// Jidien Kachu Edited in 2025/09/25
FUNCTION_BLOCK FB_WareHouseWithRobotMove_V2 EXTENDS FB_ObjectBase_V2 IMPLEMENTS IBasicElement
VAR_INPUT
    Robot     : REFERENCE TO FB_FanucRobot_Basic;
    WareHouse : REFERENCE TO FB_WareHouse;
   // Command   : ST_WareHouseWithRobotMove_Command;
    Info	  : st_AutoSixAxisWarehouseParameter;
	Stop	  : BOOL;
	//Edited by Jidien Kachu in 2025/09/25
	iSetRetryCnt	: UINT := 10;
END_VAR
VAR_OUTPUT
  // Status : ST_WareHouseWithRobotMove_Status;
END_VAR
VAR
	_Abort		: BOOL;
	strStatus	: STRING;
	uiResumeStep : UINT;
	ClampA_WareHouseCoordinates : ST_WareHouseCoordinates;
    ClampB_WareHouseCoordinates : ST_WareHouseCoordinates;
	UseA 	: BOOL;
	UseB	: BOOL;
	TargetWarehouse : E_WareHouse;
	Get 	:BOOL;
	tonTimeout		:TON;
	bTimeOutIN			   : BOOL;
	tonRobotTimeout		:TON;
	bRobotTimeoutIN			   : BOOL;
	_UniqueErrorCode :STRING;
	PreviousStrStatus : STRING;
	PreviousErrorCode : STRING;
	//Edited by Jidien Kachu in 2025/09/25
	iActRetryCnt	: UINT;
	uiBothStep : UINT;
	uiLastBothStep : UINT;
END_VAR

SUPER^.A10_StateControl();
A00_BasicUnits();

ACTION A00_BasicUnits:
tonTimeOut(IN:= bTimeOutIN AND NOT THIS^.Stop, PT:=T#30S);
tonRobotTimeout(IN:= bRobotTimeoutIN AND NOT THIS^.Stop,PT:=T#60S);
ErrorID :=2400;
END_ACTION

METHOD M_CheckCommand : BOOL // True : Command is useful
VAR_INPUT
END_VAR
VAR
	
END_VAR
// Check command paremeter is correct

IF NOT Info.Warehouse_A AND NOT Info.Warehouse_B THEN
	strStatus:='Wrong command , No warehouse selected';
	M_CheckCommand:=FALSE;
	RETURN;
ELSIF  Info.Warehouse_A AND  Info.Warehouse_B THEN
	strStatus:='Wrong command , Both warehouses selected';
	M_CheckCommand:=FALSE;
	RETURN;
ELSIF	Info.Warehouse_A THEN
	TargetWarehouse:=E_WareHouse.WareHouseA;
ELSIF	Info.Warehouse_B THEN
	TargetWarehouse:=E_WareHouse.WareHouseB;
END_IF

IF Info.Get_A <> Info.Get_B THEN
	strStatus:='Wrong command ,GetA not match to GetB';
	M_CheckCommand:=FALSE;
	RETURN;
	ELSE
		
	Get :=Info.Get_A;
END_IF


CASE LREAL_TO_INT(Info.Layer_A) OF

1,2,3,4,5,6,7,8,9,10:
	//Normal
	// Layer A in correct range
	IF ((Info.Slide_A < 1) OR (Info.Slide_A > 20)) THEN
		strStatus := 'Command error : Clamp A target slide out of range';
		M_CheckCommand:=FALSE;
		RETURN;
	ELSE
		ClampA_WareHouseCoordinates.Layer:=LREAL_TO_INT(Info.Layer_A);
		ClampA_WareHouseCoordinates.Slide:=LREAL_TO_INT(Info.Slide_A);
   
		UseA:=TRUE;	
	END_IF
	
99:
	UseA:=FALSE;
ELSE
	 strStatus := 'Command error : Clamp A target layer out of range.';
	 M_CheckCommand:=FALSE;
	 RETURN;
END_CASE


CASE LREAL_TO_INT(Info.Layer_B) OF

1,2,3,4,5,6,7,8,9,10:
//Normal
	// Layer A in correct range
	IF ((Info.Slide_B < 1) OR (Info.Slide_B > 20)) THEN
		strStatus := 'Command error : Clamp B target slide out of range';
		M_CheckCommand:=FALSE;
		RETURN;
	ELSE
		ClampB_WareHouseCoordinates.Layer:=LREAL_TO_INT(Info.Layer_B);
		ClampB_WareHouseCoordinates.Slide:=LREAL_TO_INT(Info.Slide_B);
		UseB:=TRUE;	
	END_IF
	
99:
		UseB:=FALSE;
ELSE
	 strStatus := 'Command error : Clamp B target layer out of range.';
	 M_CheckCommand:=FALSE;
	 RETURN;
END_CASE


M_CheckCommand:=TRUE;
END_METHOD

METHOD M_CheckUnitsNotBusy : BOOL
VAR_INPUT
END_VAR
M_CheckUnitsNotBusy := true;
END_METHOD

METHOD M_CheckUnitsReady : BOOL
VAR_INPUT
END_VAR
M_CheckUnitsReady := true;
END_METHOD

METHOD  M_STATE_ABORTED
VAR_INPUT
END_VAR
ERROR :=TRUE;
Busy    := FALSE;
Aborted := TRUE;
Status := strStatus;
UniqueErrorCode:=_UniqueErrorCode;
IF NOT Execute THEN
	eSTATE:=STATE_RESETTING;
END_IF

IF Execute AND Reset THEN 
	PreviousStrStatus := strStatus;
	PreviousErrorCode := _UniqueErrorCode;
	uiExecutingStep :=uiResumeStep;
	eSTATE:=STATE_EXECUTING;
	
	iActRetryCnt := iActRetryCnt + 1; //Edited by Jidien Kachu in 2025/09/25
	ERROR :=FALSE;
	Aborted := FALSE;
	uiBothStep := uiLastBothStep;
END_IF
END_METHOD

METHOD  M_STATE_ABORTING
VAR_INPUT
END_VAR
CASE uiAbortingStep OF
	0 :
		uiAbortingStep:=9999;
		bTimeOutIN:=FALSE;
		bRobotTimeoutIN :=FALSE;
		IF strStatus = PreviousStrStatus THEN
			_UniqueErrorCode :=PreviousErrorCode;
		END_IF
		_Abort :=FALSE;
		(*=====Edited by Jidien Kachu in 2025/09/25=====*)
		Robot.M_ResetAllCommand();
		WareHouse.M_ResetReloadBox();
		WareHouse.M_ResetFeedInBox();
		(*==============================================*)
	9999:	_AbortCompleted:=TRUE;
END_CASE

IF _AbortCompleted THEN	
	eSTATE :=STATE_ABORTED;
END_IF
END_METHOD

METHOD  M_STATE_DONE
VAR_INPUT
END_VAR
Busy := FALSE;
Done := TRUE;
IF NOT Execute THEN
    eState := STATE_RESETTING;
END_IF
END_METHOD

METHOD  M_STATE_DORMANT
VAR_INPUT
END_VAR
// Clear FB output
Busy            := FALSE;
Done            := FALSE;
Aborted         := FALSE;
Error           := FALSE;
ErrorID         := 0;
Status          := '';
_ResetCompleted := FALSE;
_Error          := FALSE;
_Executed       := FALSE;
strStatus :='No Error';
bTimeOutIN :=FALSE;
bRobotTimeoutIN :=FALSE;
uiExecutingStep :=uiResettingStep :=uiResumeStep :=0;
PreviousStrStatus			 :='';
PreviousErrorCode			 :='';

// Wait Execute command
IF Execute THEN
    eState := STATE_EXECUTING;
END_IF
END_METHOD

METHOD  M_STATE_ERROR
VAR_INPUT
END_VAR
ERROR   :=TRUE;
Busy	:=FALSE;
Status := strStatus;
UniqueErrorCode:=_UniqueErrorCode;
IF NOT Execute THEN	
eSTATE:=STATE_RESETTING;
END_IF
END_METHOD

METHOD  M_STATE_EXECUTING
VAR_INPUT
END_VAR
VAR_INST
	BoxReady_1st : BOOL;
	BoxReady_2nd : BOOL;  
    
    ClampA_WareHouseCoordinates : ST_WareHouseCoordinates;
    ClampB_WareHouseCoordinates : ST_WareHouseCoordinates;
	

	
END_VAR
VAR
	
END_VAR
// Set Busy active edit by johnson
Busy := TRUE;
(*IF THIS^.Stop THEN // Pending the timeout when Stop signal occur
	bTimeOutIN :=FALSE;
	bRobotTimeoutIN :=FALSE;
END_IF*)
// Service Process
CASE uiExecutingStep OF
	0:
        // Clear variable
       
        bTimeOutIN :=FALSE;
//        uiBothStep := 0;
		uiLastBothStep := 0; //Edited by Jidien Kachu in 2025/10/09
		BoxReady_1st := 0;
		BoxReady_2nd := 0;
        // Check command
        IF M_CheckCommand() THEN
            uiExecutingStep := 10;
		ELSE
			_Error:=TRUE;
        END_IF
		iActRetryCnt := 0; //Edited by Jidien Kachu in 2025/09/25
    10:
        // Start process, check units first
        IF M_CheckUnitsReady() THEN
            uiExecutingStep := 20;
        END_IF
    20:
        // CHeck units not busy state
        IF M_CheckUnitsNotBusy() THEN
            uiExecutingStep := 1000;
        END_IF
   
	1000:   
			// Read  Warehouse coordinate
			ClampA_WareHouseCoordinates := THIS^.ClampA_WareHouseCoordinates;
            ClampB_WareHouseCoordinates := THIS^.ClampB_WareHouseCoordinates;     
			IF UseA AND NOT UseB THEN
				//Only clampA
				uiExecutingStep := 10000;
			ELSIF NOT UseA AND UseB THEN
				//Only ClampB 
				uiExecutingStep := 20000;
			ELSIF UseA AND UseB THEN
				//Both Clamps
				uiExecutingStep := 30000;		
			END_IF
       
    10000: // Only ClampA 
        IF NOT Robot._DI1.Done THEN
            // Read ClampA Warehouse coordinate
            ClampA_WareHouseCoordinates := THIS^.ClampA_WareHouseCoordinates;
			
			IF Get THEN// Prepare Box
				//Pick Box
				 WareHouse.M_StartReloadBox(WareHouseSelect := TargetWarehouse, WarehouseCoordinates := ClampA_WareHouseCoordinates);

           		 // Check Box reload completed
           		 IF WareHouse.bReloadBox_Completed THEN
           	     BoxReady_1st := TRUE;
          		  END_IF
				  // Robot Warehouse move
           		 Robot.M_StartWareHousePickUpBox_ClampA(WareHouseSelect := TargetWarehouse,
                                                   Info            := ClampA_WareHouseCoordinates,
                                                   BoxReady_1st    := BoxReady_1st);
//				bTimeOutIN:=TRUE;
				IF tonTimeout.Q THEN
					_Error:=TRUE;
					strStatus:='Clamp A reolad box timeout';
				END_IF
				  
			ELSE
					//Place Box
					WareHouse.M_StartFeedInBox(WareHouseSelect := TargetWarehouse, WarehouseCoordinates := ClampA_WareHouseCoordinates);

           			 // Check Box reload completed
           			 IF WareHouse.bFeedInBox_Completed THEN
               			 BoxReady_1st := TRUE;
          		 	 END_IF				
					           
			 	Robot.M_StartWareHousePlaceBox_ClampA(WareHouseSelect := TargetWarehouse,
                                                   Info            := ClampA_WareHouseCoordinates,
                                                   BoxReady_1st    := BoxReady_1st);
            	
//				bTimeOutIN:=TRUE;
				IF tonTimeout.Q THEN
					_Error:=TRUE;
					strStatus:='Clamp A Feedin box timeout';
				END_IF
           END_IF
        ELSE
            uiExecutingStep := 10080;
        END_IF
		
		bRobotTimeoutIN :=TRUE;
		IF tonRobotTimeout.Q THEN
			(*=====Edited by Jidien Kachu in 2025/09/25=====*)
			IF iActRetryCnt = iSetRetryCnt THEN
				_Error:=TRUE;
			ELSE
				_Abort := TRUE;
				uiAbortingStep := 0;
			END_IF
			
			(*==============================================*)
			strStatus:='Clamp A  robot timeout';
		END_IF
		
    10080:
        Robot.M_ResetAllCommand(); // Clear command and go to place box
		bTimeOutIN :=FALSE;
		bRobotTimeoutIN :=FALSE;
        IF NOT Robot._DI1.Done THEN
            uiExecutingStep := 99000; 
        END_IF
    
    
   20000: // Only ClampB
        IF NOT Robot._DI1.Done THEN
            			
			IF Get THEN// Prepare Box
				//Pick Box
				 WareHouse.M_StartReloadBox(WareHouseSelect := TargetWarehouse, WarehouseCoordinates := ClampB_WareHouseCoordinates);

           		 // Check Box reload completed
           		 IF WareHouse.bReloadBox_Completed THEN
           	     BoxReady_2nd := TRUE;
          		  END_IF
				  // Robot Warehouse move
           		 Robot.M_StartWareHousePickUpBox_ClampB(WareHouseSelect := TargetWarehouse,
                                                   Info            := ClampB_WareHouseCoordinates,
                                                   BoxReady_2nd    := BoxReady_2nd);

//				bTimeOutIN:=TRUE;
				IF tonTimeout.Q THEN
					_Error:=TRUE;
					strStatus:='Clamp B Reload box timeout';
				END_IF
			ELSE
					//Place Box
					WareHouse.M_StartFeedInBox(WareHouseSelect := TargetWarehouse, WarehouseCoordinates := ClampB_WareHouseCoordinates);

           			 // Check Box reload completed
           			 IF WareHouse.bFeedInBox_Completed THEN
               			 BoxReady_2nd := TRUE;
          		 	 END_IF				
					           
			 	Robot.M_StartWareHousePlaceBox_ClampB (WareHouseSelect := TargetWarehouse,
                                                   Info            := ClampB_WareHouseCoordinates,
                                                   BoxReady_2nd    := BoxReady_2nd);
//            	bTimeOutIN:=TRUE;
				IF tonTimeout.Q THEN
					_Error:=TRUE;
					strStatus:='Clamp B Feedin box timeout';
				END_IF
           END_IF
        ELSE
            uiExecutingStep := 20080;
        END_IF
		
		bRobotTimeoutIN :=TRUE;
		IF tonRobotTimeout.Q THEN
			(*=====Edited by Jidien Kachu in 2025/09/25=====*)
			IF iActRetryCnt = iSetRetryCnt THEN
				_Error:=TRUE;
			ELSE
				_Abort := TRUE;
				uiAbortingStep := 0;
			END_IF
			(*==============================================*)
			strStatus:='Clamp B Robot timeout';
		END_IF
		
    20080:
        Robot.M_ResetAllCommand(); // Clear command and go to place box
		bTimeOutIN :=FALSE;
		bRobotTimeoutIN :=FALSE;

        IF NOT Robot._DI1.Done THEN
            uiExecutingStep := 99000; 
        END_IF
		
    30000: // Both Clamps
        		
		IF Get THEN //BOth clamps pick
        CASE uiBothStep OF
            0: // ClampA target slide move the box to front side
                WareHouse.M_StartReloadBox(WareHouseSelect      := TargetWarehouse,
                                           WarehouseCoordinates := ClampA_WareHouseCoordinates);
				
				bTimeOutIN :=TRUE;
				IF tonTimeout.Q THEN
					(*=====Edited by Jidien Kachu in 2025/09/25=====*)
					IF iActRetryCnt = iSetRetryCnt THEN
						_Error:=TRUE;
					ELSE
						_Abort := TRUE;
						uiAbortingStep := 0;
					END_IF
					(*==============================================*)
					strStatus:='Clamp A reload timeout';
				END_IF
               
                IF WareHouse.bReloadBox_Completed THEN
					bTimeOutIN :=FALSE;
                    BoxReady_1st     := TRUE;
                    uiBothStep := 10;
                END_IF

            10: // wait Robot Allow continue
			 		WareHouse.M_ResetReloadBox();
                IF Robot._DI1.Notification // AND
//                    NOT
//                    WareHouse._stWarehouseList.ASide_Layers[ClampA_WareHouseCoordinates.Layer].stStatus.bSlides[ClampA_WareHouseCoordinates.Slide]
                    THEN
                   
					
                    IF NOT WareHouse.bReloadBox_Completed THEN					
               
                        uiBothStep := 15;
                    END_IF

                END_IF
			15:	IF NOT WareHouse._stWarehouseList.ASide_Layers[ClampA_WareHouseCoordinates.Layer].stStatus.bSlides[ClampA_WareHouseCoordinates.Slide] THEN
					 uiBothStep := 20;	
				 END_IF
				 
            20: // ClampB target slide move the box to front slide
                WareHouse.M_StartReloadBox(WareHouseSelect := TargetWarehouse, WarehouseCoordinates := ClampB_WareHouseCoordinates);
				bTimeOutIN :=TRUE;
                IF WareHouse.bReloadBox_Completed THEN
					bTimeOutIN :=FALSE;
                    BoxReady_2nd     := TRUE;
                    uiBothStep := 99;
                END_IF
				IF tonTimeout.Q THEN
					(*=====Edited by Jidien Kachu in 2025/09/25=====*)
					IF iActRetryCnt = iSetRetryCnt THEN
						_Error:=TRUE;
					ELSE
						_Abort := TRUE;
						uiAbortingStep := 0;
						uiLastBothStep := 20;
					END_IF
					(*==============================================*)
					strStatus:='Clamp B reload timeout';
				END_IF
				
				
            99:
				WareHouse.M_ResetReloadBox();
        // wait reset
        END_CASE

        Robot.M_StartWareHousePickUpBox_ClampBoth(WareHouseSelect := TargetWarehouse,
                                                  ClampA_Info     := ClampA_WareHouseCoordinates,
                                                  ClampB_Info     := ClampB_WareHouseCoordinates,
                                                  BoxReady_1st    := BoxReady_1st,
                                                  BoxReady_2nd    := BoxReady_2nd);
												  
		bRobotTimeoutIN :=TRUE;
		IF tonRobotTimeout.Q THEN
			(*=====Edited by Jidien Kachu in 2025/09/25=====*)
			IF iActRetryCnt = iSetRetryCnt THEN
				_Error:=TRUE;
			ELSE
				_Abort := TRUE;
				uiAbortingStep := 0;
			END_IF
			(*==============================================*)
			strStatus:='Robot timeout';
		END_IF
		ELSE
		  CASE uiBothStep OF
			  
			   0: // ClampA target slide move the box to front side
                WareHouse.M_StartFeedInBox(WareHouseSelect      := TargetWarehouse,
                                           WarehouseCoordinates := ClampA_WareHouseCoordinates);

               bTimeOutIN :=TRUE;
                IF WareHouse.bFeedInBox_Completed THEN
					bTimeOutIN :=FALSE;
                    BoxReady_1st     := TRUE;
                    uiBothStep := 10;
                END_IF
				IF tonTimeout.Q THEN
					(*=====Edited by Jidien Kachu in 2025/09/25=====*)
					IF iActRetryCnt = iSetRetryCnt THEN
						_Error:=TRUE;
					ELSE
						_Abort := TRUE;
						uiAbortingStep := 0;
					END_IF
					(*==============================================*)
					strStatus:='Clamp A Feedin timeout';
				END_IF

            10: // wait Robot Allow continue
					WareHouse.M_ResetFeedInBox();
                 IF Robot._DI1.Notification //AND
                     
//                    WareHouse._stWarehouseList.ASide_Layers[ClampA_WareHouseCoordinates.Layer].stStatus.bSlides[ClampA_WareHouseCoordinates.Slide]
                    THEN
                    

                    IF NOT WareHouse.bFeedInBox_Completed THEN
                        uiBothStep := 15;
                    END_IF

                END_IF
			15:  
				uiBothStep := 20;
			
            20: // ClampB target slide move the box to front slide
                WareHouse.M_StartFeedInBox(WareHouseSelect := TargetWarehouse, WarehouseCoordinates := ClampB_WareHouseCoordinates);
				bTimeOutIN :=TRUE;
                IF WareHouse.bFeedInBox_Completed THEN
					bTimeOutIN :=FALSE;
                    BoxReady_2nd     := TRUE;
                    uiBothStep := 99;
                END_IF
				IF tonTimeout.Q THEN
					(*=====Edited by Jidien Kachu in 2025/09/25=====*)
					IF iActRetryCnt = iSetRetryCnt THEN
						_Error:=TRUE;
					ELSE
						_Abort := TRUE;
						uiAbortingStep := 0;
						uiLastBothStep := 20;
					END_IF
					(*==============================================*)
					strStatus:='Clamp B Feedin timeout';
				END_IF
            99: 
				WareHouse.M_ResetFeedInBox();

        END_CASE

        Robot.M_StartWareHousePlaceUpBox_ClampBoth(WareHouseSelect := TargetWarehouse,
                                                  ClampA_Info     := ClampA_WareHouseCoordinates,
                                                  ClampB_Info     := ClampB_WareHouseCoordinates,
                                                  BoxReady_1st    := BoxReady_1st,
                                                  BoxReady_2nd    := BoxReady_2nd);
												  
		bRobotTimeoutIN :=TRUE;
			IF tonRobotTimeout.Q THEN
				(*=====Edited by Jidien Kachu in 2025/09/25=====*)
				IF iActRetryCnt = iSetRetryCnt THEN
					_Error:=TRUE;
				ELSE
					_Abort := TRUE;
					uiAbortingStep := 0;
				END_IF
				(*==============================================*)
				strStatus:='Robot timeout';
			END_IF
		END_IF
		
        IF Robot._DI1.Done THEN
			uiBothStep := 0;
            uiExecutingStep := 30080;
        END_IF
		
    30080: // Check robot command is clear
        WareHouse.M_ResetReloadBox();
        WareHouse.M_ResetFeedInBox();
        Robot.M_ResetAllCommand();
		bTimeOutIN :=FALSE;
		bRobotTimeoutIN :=FALSE;
		
        IF NOT Robot._DI1.Done THEN
            uiExecutingStep := 99000; // go to place step
        END_IF    
   
   
    99000: // process done
                Status    := 'Process completed';
        _Executed := TRUE;
END_CASE
IF _Executed THEN
    eState := STATE_DONE;
ELSIF _Error THEN
	//FUN_UniqueErrorCodeGenerator(iErrorID := ErrorID,UinqueErrorCode=>_UniqueErrorCode);
    eState := STATE_ERROR;
ELSIF NOT Execute THEN
    eState := STATE_RESETTING;
END_IF
IF _Abort OR Abort THEN
	//FUN_UniqueErrorCodeGenerator(iErrorID := ErrorID,UinqueErrorCode=>_UniqueErrorCode);
	eSTATE:=STATE_ABORTING;
END_IF
END_METHOD

METHOD  M_STATE_RESETTING
VAR_INPUT
END_VAR
Error :=FALSE;
Done :=FALSE;
Busy := FALSE;
_Error :=FALSE;

CASE uiResettingStep OF
	
	0:
		bTimeOutIN :=FALSE;
		bRobotTimeoutIN :=FALSE;
		Robot.M_ResetAllCommand();
		uiResettingStep:=9999;
		WareHouse.M_ResetFeedInBox();
		WareHouse.M_ResetReloadBox();
	9999:
		_ResetCompleted:=TRUE;
END_CASE
IF _ResetCompleted THEN
	eSTATE:=STATE_DORMANT;
END_IF
END_METHOD

END_FUNCTION_BLOCK

(* stored: Version 1.1.0.1, ProductVersion 3.1.4024.13
   POU FB_WareHouseWithRobotMove_V2: Id {b288e5e4-52bf-4254-a560-b7f47a4ab827}, SpecialFunc None
   Folder Method: Id {7da9048b-1ed4-4cc1-a9b9-7d5d0bdf0516}
   Folder State: Id {055e6999-d74e-42a2-8e38-c39d00df113d}
   Action A00_BasicUnits: Id {d23b4903-f81c-4cd2-94a4-fe7fa85cc4ba}
   Method M_CheckCommand: Id {63515dfa-5411-48ba-b30e-a291ffce2619}
   Method M_CheckUnitsNotBusy: Id {63eed7d5-41c9-4063-a407-a9bd703c4e64}
   Method M_CheckUnitsReady: Id {1f8f0145-58c9-4c6c-80ee-5bf58e29a38f}
   Method M_STATE_ABORTED: Id {c448e92d-f3c1-4066-a9bc-7495cd087342}
   Method M_STATE_ABORTING: Id {d782a69f-50e7-4e5a-a67e-f157af942c87}
   Method M_STATE_DONE: Id {e34bcbf6-3a9b-4bdb-b87b-90d195630ca2}
   Method M_STATE_DORMANT: Id {d13610a9-98cf-4d7e-8b9a-1781c145229e}
   Method M_STATE_ERROR: Id {38b2cd84-5930-42d4-832d-815a2540b20c}
   Method M_STATE_EXECUTING: Id {d8a0c167-8a74-46d1-9eb1-057c4bf761a0}
   Method M_STATE_RESETTING: Id {64342353-f3e1-4a9a-a45b-35126dcdc89f} *)
